SUBAPPLICATION Uebung_010b4 (* SoftKey_F1-8 auf DigitalOutput_Q1-8 *)
  (* Standard: 61499-2; Description: Copyright (c) 2023 Meisterschulen am Ostbahnhof This program and the accompanying materials are made available under the terms of the Eclipse Public License 2.0 which is available at https://www.eclipse.org/legal/epl-2.0/ SPDX-License-Identifier: EPL-2.0 *)
  (* Version 1.0, 2023-10-23, Franz Höpfinger, Meisterschulen am Ostbahnhof *)
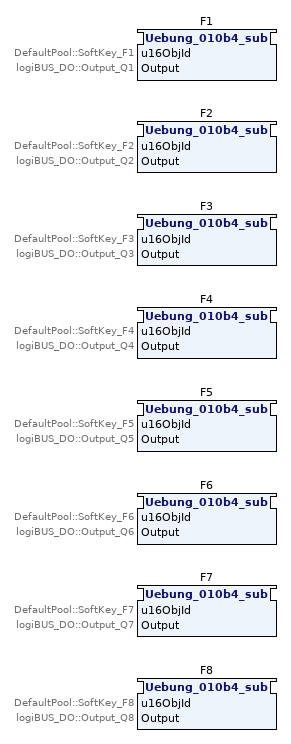
  SUBAPPS
    F1 : Uebung_010b4_sub(u16ObjId := DefaultPool::SoftKey_F1, Output := logiBUS_DO::Output_Q1);
    F2 : Uebung_010b4_sub(u16ObjId := DefaultPool::SoftKey_F2, Output := logiBUS_DO::Output_Q2);
    F3 : Uebung_010b4_sub(u16ObjId := DefaultPool::SoftKey_F3, Output := logiBUS_DO::Output_Q3);
    F4 : Uebung_010b4_sub(u16ObjId := DefaultPool::SoftKey_F4, Output := logiBUS_DO::Output_Q4);
    F5 : Uebung_010b4_sub(u16ObjId := DefaultPool::SoftKey_F5, Output := logiBUS_DO::Output_Q5);
    F6 : Uebung_010b4_sub(u16ObjId := DefaultPool::SoftKey_F6, Output := logiBUS_DO::Output_Q6);
    F7 : Uebung_010b4_sub(u16ObjId := DefaultPool::SoftKey_F7, Output := logiBUS_DO::Output_Q7);
    F8 : Uebung_010b4_sub(u16ObjId := DefaultPool::SoftKey_F8, Output := logiBUS_DO::Output_Q8);
  END_SUBAPPS
END_SUBAPPLICATION
